RoboDK station: 6640_station_curve1.rdk

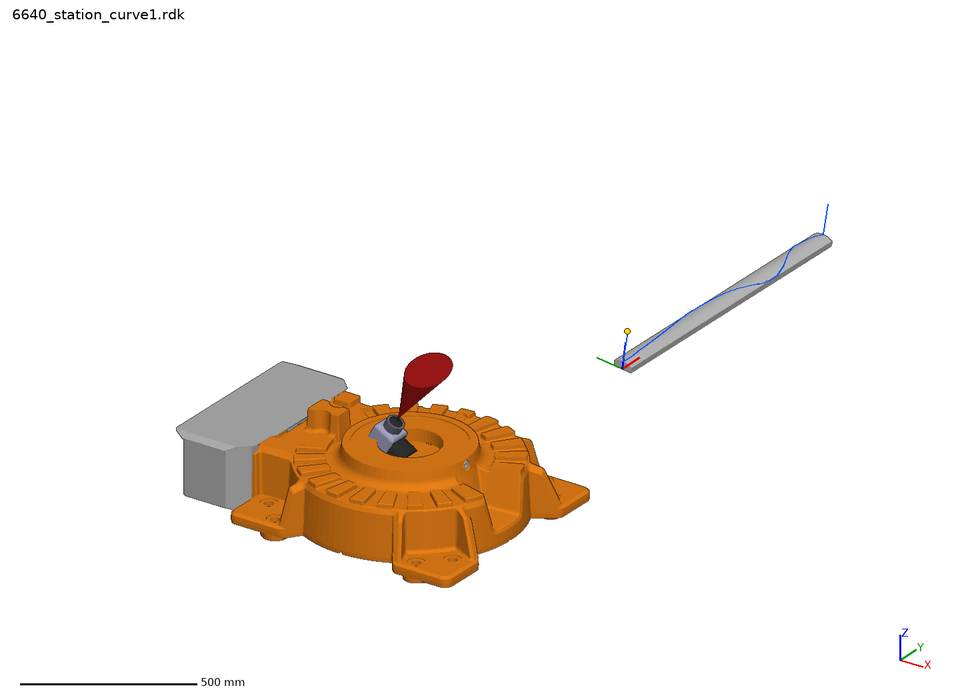
[picture v0: the station drawn from its stored meshes, robots at their saved joint values, targets as dots, program paths as lines]
Station 6640_station_curve1 (saved by RoboDK 5.3.2). Poses are relative to the parent item; angles as X-Y-Z fixed-axis rotations.
  - frame Frame 3 at (1086.51, -506.82, 968.91) mm, rotated rx 8.27 ry 0.16 rz 90.47 deg
    - object Curve_sparse at (0, 0, 0) mm
    - object wood at (0, 0, 0) mm, size 1000 x 60 x 25.4 mm, geometry from wood.stl
  - machining project Path1 settings: rotZ(0) | rotX(0)*rotY(0) | rotz(0)
  - program Path1 (113 instructions, listed below)
  - robot ABB IRB 6640-180/2.55: 6 axes, payload 180 kg, reach 2550 mm, repeatability 0.07 mm, weight 1310 kg
      joint limits [-170, -65, -180, -300, -120, -360] to [170, 85, 70, 300, 120, 360]; home [0, 0, 0, 0, 0, 0]; saved at [28.636, -24.413, 34.192, -11.874, 61.538, 32.546]
    - tool Paint gun, TCP at (75, 0, 493.3) mm, rotated rx 0 ry 30 rz 0 deg, size 203.2 x 279.7 x 471.5 mm
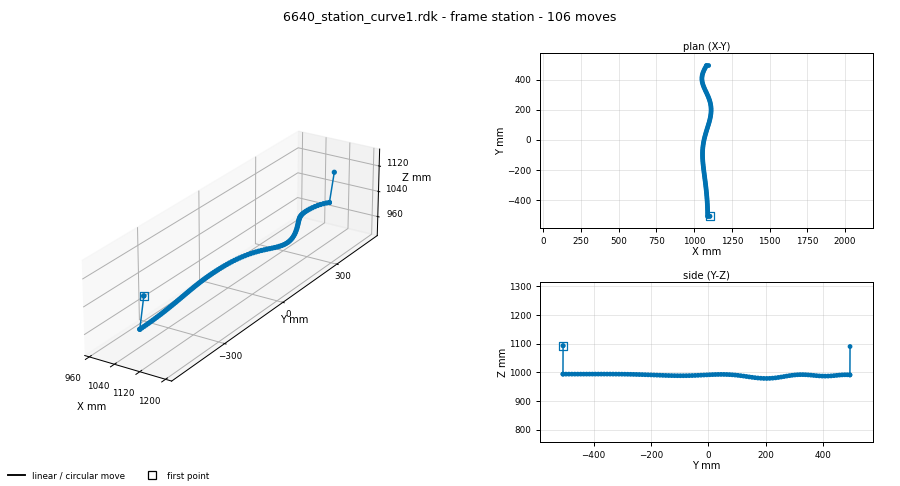
[picture p0: tool path of 6640_station_curve1.rdk in frame station, 106 of 106 moves have a stored position in this frame; points joined in program order, loops and branches not executed]

--- program Path1 (robot ABB IRB 6640-180/2.55) ---
  Smooth(1)
  Set speed (500.0 mm/s)
  Set Ref.: Frame 3
  Set Tool: Paint gun
  Show Paint gun
  MoveJ 1 to (0, 0, 125.4) mm, rotated rx 180 ry 0 rz 89.52 deg; joints [-28.763, -23.766, 33.648, 11.507, 61.252, -32.677]
  MoveL 2 to (0, 0, 125.4) mm, rotated rx 180 ry 0 rz 89.52 deg; joints [-28.763, -23.766, 33.648, 11.507, 61.252, -32.677]
  MoveL 3 to (0, 0, 25.4) mm, rotated rx 180 ry 0 rz 89.52 deg; joints [-29.166, -24.266, 38.853, 12.236, 56.729, -34.255]
  MoveL 4 to (0, 0, 25.4) mm, rotated rx 180 ry 0 rz 89.52 deg; joints [-29.166, -24.266, 38.853, 12.236, 56.729, -34.255]
  Set speed (50.0 mm/s)
  MoveL 5 to (10.27, 0.03, 25.4) mm, rotated rx 180 ry 0.03 rz 89.52 deg; joints [-28.68, -24.594, 39.061, 12.062, 56.719, -33.688]
  MoveL 6 to (20.55, 0.12, 25.4) mm, rotated rx 180 ry 0.13 rz 89.52 deg; joints [-28.212, -24.963, 39.304, 11.937, 56.664, -33.163]
  MoveL 7 to (30.82, 0.27, 25.4) mm, rotated rx 180 ry 0.3 rz 89.52 deg; joints [-27.761, -25.373, 39.58, 11.859, 56.565, -32.678]
  MoveL 8 to (41.1, 0.48, 25.4) mm, rotated rx 180 ry 0.54 rz 89.52 deg; joints [-27.327, -25.825, 39.89, 11.827, 56.42, -32.233]
  MoveL 9 to (51.37, 0.75, 25.39) mm, rotated rx 179.99 ry 0.84 rz 89.52 deg; joints [-26.908, -26.32, 40.233, 11.838, 56.23, -31.825]
  MoveL 10 to (61.65, 1.07, 25.39) mm, rotated rx 179.99 ry 1.21 rz 89.52 deg; joints [-26.505, -26.859, 40.611, 11.891, 55.993, -31.454]
  MoveL 11 to (71.92, 1.46, 25.38) mm, rotated rx 179.99 ry 1.65 rz 89.52 deg; joints [-26.116, -27.442, 41.023, 11.986, 55.711, -31.119]
  MoveL 12 to (82.18, 1.91, 25.36) mm, rotated rx 179.98 ry 2.15 rz 89.52 deg; joints [-25.741, -28.07, 41.469, 12.121, 55.383, -30.819]
  MoveL 13 to (92.45, 2.41, 25.34) mm, rotated rx 179.98 ry 2.72 rz 89.52 deg; joints [-25.379, -28.743, 41.949, 12.295, 55.009, -30.552]
  MoveL 14 to (102.71, 2.98, 25.31) mm, rotated rx 179.97 ry 3.35 rz 89.52 deg; joints [-25.03, -29.461, 42.464, 12.507, 54.591, -30.32]
  MoveL 15 to (112.97, 3.6, 25.27) mm, rotated rx 179.97 ry 4.05 rz 89.52 deg; joints [-24.692, -30.224, 43.013, 12.756, 54.127, -30.119]
  MoveL 16 to (123.22, 4.28, 25.22) mm, rotated rx 179.96 ry 4.81 rz 89.52 deg; joints [-24.365, -31.033, 43.595, 13.042, 53.621, -29.95]
  MoveL 17 to (133.47, 5.01, 25.15) mm, rotated rx 179.95 ry 5.64 rz 89.52 deg; joints [-24.047, -31.886, 44.21, 13.362, 53.072, -29.811]
  MoveL 18 to (143.72, 5.8, 25.07) mm, rotated rx 179.95 ry 6.52 rz 89.52 deg; joints [-23.737, -32.783, 44.857, 13.716, 52.483, -29.701]
  MoveL 19 to (153.96, 6.65, 24.97) mm, rotated rx 179.94 ry 7.45 rz 89.52 deg; joints [-23.435, -33.723, 45.536, 14.101, 51.854, -29.619]
  MoveL 20 to (164.2, 7.54, 24.84) mm, rotated rx 179.93 ry 8.44 rz 89.52 deg; joints [-23.137, -34.705, 46.244, 14.515, 51.19, -29.561]
  MoveL 21 to (174.44, 8.49, 24.69) mm, rotated rx 179.92 ry 9.48 rz 89.52 deg; joints [-22.843, -35.726, 46.981, 14.956, 50.491, -29.527]
  MoveL 22 to (184.66, 9.48, 24.52) mm, rotated rx 179.91 ry 10.57 rz 89.52 deg; joints [-22.55, -36.783, 47.743, 15.421, 49.762, -29.511]
  MoveL 23 to (194.89, 10.51, 24.31) mm, rotated rx 179.9 ry 11.69 rz 89.51 deg; joints [-22.256, -37.875, 48.528, 15.904, 49.006, -29.511]
  MoveL 24 to (205.11, 11.59, 24.08) mm, rotated rx 179.89 ry 12.85 rz 89.51 deg; joints [-21.959, -38.997, 49.334, 16.402, 48.225, -29.522]
  MoveL 25 to (215.32, 12.7, 23.81) mm, rotated rx 179.88 ry 14.03 rz 89.51 deg; joints [-21.654, -40.146, 50.156, 16.908, 47.426, -29.538]
  MoveL 26 to (225.53, 13.84, 23.52) mm, rotated rx 179.87 ry 15.24 rz 89.5 deg; joints [-21.34, -41.317, 50.991, 17.415, 46.611, -29.552]
  MoveL 27 to (235.73, 15, 23.18) mm, rotated rx 179.86 ry 16.45 rz 89.5 deg; joints [-21.012, -42.505, 51.834, 17.916, 45.786, -29.557]
  MoveL 28 to (245.94, 16.19, 22.82) mm, rotated rx 179.85 ry 17.68 rz 89.5 deg; joints [-20.667, -43.704, 52.681, 18.4, 44.955, -29.543]
  MoveL 29 to (256.14, 17.39, 22.42) mm, rotated rx 179.83 ry 18.9 rz 89.49 deg; joints [-20.301, -44.909, 53.526, 18.858, 44.122, -29.502]
  MoveL 30 to (266.33, 18.6, 22) mm, rotated rx 179.82 ry 20.1 rz 89.48 deg; joints [-19.91, -46.112, 54.365, 19.278, 43.293, -29.422]
  MoveL 31 to (276.53, 19.8, 21.54) mm, rotated rx 179.81 ry 21.29 rz 89.48 deg; joints [-19.49, -47.308, 55.191, 19.646, 42.473, -29.291]
  MoveL 32 to (286.73, 20.99, 21.06) mm, rotated rx 179.8 ry 22.45 rz 89.47 deg; joints [-19.036, -48.488, 55.998, 19.951, 41.665, -29.097]
  MoveL 33 to (296.93, 22.16, 20.57) mm, rotated rx 179.79 ry 23.56 rz 89.46 deg; joints [-18.546, -49.644, 56.78, 20.176, 40.876, -28.827]
  MoveL 34 to (307.13, 23.29, 20.06) mm, rotated rx 179.77 ry 24.63 rz 89.46 deg; joints [-18.015, -50.768, 57.531, 20.307, 40.109, -28.466]
  MoveL 35 to (317.34, 24.39, 19.55) mm, rotated rx 179.76 ry 25.64 rz 89.45 deg; joints [-17.44, -51.851, 58.245, 20.331, 39.37, -28.002]
  MoveL 36 to (327.55, 25.42, 19.04) mm, rotated rx 179.75 ry 26.59 rz 89.44 deg; joints [-16.818, -52.883, 58.914, 20.231, 38.664, -27.422]
  MoveL 37 to (337.77, 26.39, 18.54) mm, rotated rx 179.74 ry 27.45 rz 89.43 deg; joints [-16.146, -53.855, 59.534, 19.995, 37.996, -26.713]
  MoveL 38 to (348, 27.28, 18.08) mm, rotated rx 179.73 ry 28.23 rz 89.43 deg; joints [-15.422, -54.756, 60.096, 19.611, 37.374, -25.864]
  MoveL 39 to (358.24, 28.06, 17.65) mm, rotated rx 179.72 ry 28.92 rz 89.42 deg; joints [-14.647, -55.574, 60.594, 19.07, 36.803, -24.867]
  MoveL 40 to (368.48, 28.74, 17.27) mm, rotated rx 179.71 ry 29.5 rz 89.41 deg; joints [-13.819, -56.299, 61.021, 18.363, 36.293, -23.717]
  MoveL 41 to (378.74, 29.28, 16.96) mm, rotated rx 179.71 ry 29.96 rz 89.41 deg; joints [-12.939, -56.917, 61.371, 17.488, 35.851, -22.41]
  MoveL 42 to (389.01, 29.69, 16.73) mm, rotated rx 179.7 ry 30.3 rz 89.41 deg; joints [-12.01, -57.416, 61.637, 16.448, 35.489, -20.948]
  MoveL 43 to (399.28, 29.93, 16.58) mm, rotated rx 179.7 ry 30.5 rz 89.4 deg; joints [-11.036, -57.782, 61.81, 15.249, 35.219, -19.34]
  MoveL 44 to (409.55, 30, 16.54) mm, rotated rx 179.7 ry 30.56 rz 89.4 deg; joints [-10.021, -58.003, 61.885, 13.906, 35.051, -17.599]
  MoveL 45 to (419.82, 29.88, 16.61) mm, rotated rx 179.7 ry 30.46 rz 89.41 deg; joints [-8.971, -58.064, 61.852, 12.439, 35, -15.743]
  MoveL 46 to (430.09, 29.55, 16.8) mm, rotated rx 179.7 ry 30.19 rz 89.41 deg; joints [-7.893, -57.953, 61.705, 10.874, 35.08, -13.798]
  MoveL 47 to (440.35, 29.02, 17.11) mm, rotated rx 179.71 ry 29.73 rz 89.41 deg; joints [-6.798, -57.657, 61.436, 9.247, 35.305, -11.795]
  MoveL 48 to (450.59, 28.26, 17.54) mm, rotated rx 179.72 ry 29.08 rz 89.42 deg; joints [-5.695, -57.164, 61.038, 7.597, 35.69, -9.772]
  MoveL 49 to (460.8, 27.26, 18.08) mm, rotated rx 179.73 ry 28.22 rz 89.43 deg; joints [-4.595, -56.464, 60.503, 5.966, 36.248, -7.769]
  MoveL 50 to (470.99, 26.04, 18.73) mm, rotated rx 179.74 ry 27.14 rz 89.44 deg; joints [-3.511, -55.548, 59.823, 4.398, 36.992, -5.826]
  MoveL 51 to (481.13, 24.57, 19.46) mm, rotated rx 179.76 ry 25.81 rz 89.45 deg; joints [-2.455, -54.409, 58.994, 2.935, 37.931, -3.981]
  MoveL 52 to (491.24, 22.88, 20.25) mm, rotated rx 179.78 ry 24.24 rz 89.46 deg; joints [-1.438, -53.042, 58.011, 1.613, 39.076, -2.269]
  MoveL 53 to (501.3, 20.95, 21.08) mm, rotated rx 179.8 ry 22.41 rz 89.47 deg; joints [-0.471, -51.445, 56.869, 0.461, 40.433, -0.718]
  MoveL 54 to (511.32, 18.81, 21.92) mm, rotated rx 179.82 ry 20.31 rz 89.48 deg; joints [0.435, -49.618, 55.569, -0.501, 42.005, 0.656]
  MoveL 55 to (521.29, 16.45, 22.74) mm, rotated rx 179.84 ry 17.95 rz 89.49 deg; joints [1.274, -47.568, 54.113, -1.264, 43.792, 1.842]
  MoveL 56 to (531.21, 13.91, 23.5) mm, rotated rx 179.87 ry 15.31 rz 89.5 deg; joints [2.039, -45.304, 52.508, -1.827, 45.788, 2.841]
  MoveL 57 to (541.1, 11.19, 24.17) mm, rotated rx 179.9 ry 12.42 rz 89.51 deg; joints [2.729, -42.844, 50.769, -2.202, 47.981, 3.663]
  MoveL 58 to (550.95, 8.31, 24.72) mm, rotated rx 179.92 ry 9.29 rz 89.52 deg; joints [3.344, -40.212, 48.912, -2.407, 50.351, 4.325]
  MoveL 59 to (560.77, 5.31, 25.12) mm, rotated rx 179.95 ry 5.96 rz 89.52 deg; joints [3.888, -37.44, 46.967, -2.465, 52.868, 4.848]
  MoveL 60 to (570.57, 2.2, 25.35) mm, rotated rx 179.98 ry 2.48 rz 89.52 deg; joints [4.366, -34.57, 44.964, -2.402, 55.495, 5.259]
  MoveL 61 to (580.34, -0.98, 25.39) mm, rotated rx -179.99 ry -1.1 rz 89.52 deg; joints [4.789, -31.65, 42.942, -2.246, 58.183, 5.584]
  MoveL 62 to (590.1, -4.2, 25.23) mm, rotated rx -179.96 ry -4.72 rz 89.51 deg; joints [5.165, -28.732, 40.94, -2.022, 60.883, 5.846]
  MoveL 63 to (599.85, -7.41, 24.86) mm, rotated rx -179.93 ry -8.3 rz 89.5 deg; joints [5.506, -25.87, 39, -1.753, 63.536, 6.068]
  MoveL 64 to (609.6, -10.59, 24.3) mm, rotated rx -179.89 ry -11.78 rz 89.48 deg; joints [5.821, -23.114, 37.155, -1.457, 66.093, 6.268]
  MoveL 65 to (619.37, -13.69, 23.55) mm, rotated rx -179.86 ry -15.08 rz 89.46 deg; joints [6.122, -20.509, 35.436, -1.148, 68.506, 6.46]
  MoveL 66 to (629.17, -16.67, 22.66) mm, rotated rx -179.83 ry -18.17 rz 89.44 deg; joints [6.415, -18.095, 33.866, -0.838, 70.734, 6.655]
  MoveL 67 to (639.01, -19.48, 21.66) mm, rotated rx -179.79 ry -20.98 rz 89.42 deg; joints [6.709, -15.901, 32.46, -0.535, 72.747, 6.861]
  MoveL 68 to (648.9, -22.07, 20.6) mm, rotated rx -179.76 ry -23.49 rz 89.39 deg; joints [7.008, -13.952, 31.228, -0.246, 74.52, 7.085]
  MoveL 69 to (658.85, -24.39, 19.54) mm, rotated rx -179.73 ry -25.65 rz 89.37 deg; joints [7.32, -12.263, 30.174, 0.025, 76.036, 7.329]
  MoveL 70 to (668.88, -26.39, 18.55) mm, rotated rx -179.7 ry -27.45 rz 89.34 deg; joints [7.647, -10.852, 29.3, 0.271, 77.285, 7.599]
  MoveL 71 to (679, -28, 17.68) mm, rotated rx -179.67 ry -28.86 rz 89.32 deg; joints [7.995, -9.73, 28.609, 0.488, 78.253, 7.898]
  MoveL 72 to (689.18, -29.17, 17.03) mm, rotated rx -179.65 ry -29.86 rz 89.3 deg; joints [8.367, -8.911, 28.103, 0.669, 78.931, 8.23]
  MoveL 73 to (699.43, -29.84, 16.63) mm, rotated rx -179.64 ry -30.43 rz 89.29 deg; joints [8.769, -8.409, 27.786, 0.807, 79.306, 8.6]
  MoveL 74 to (709.7, -29.98, 16.55) mm, rotated rx -179.64 ry -30.55 rz 89.29 deg; joints [9.204, -8.24, 27.664, 0.891, 79.366, 9.014]
  MoveL 75 to (719.96, -29.55, 16.8) mm, rotated rx -179.65 ry -30.19 rz 89.3 deg; joints [9.679, -8.417, 27.747, 0.909, 79.097, 9.481]
  MoveL 76 to (730.17, -28.55, 17.38) mm, rotated rx -179.66 ry -29.33 rz 89.31 deg; joints [10.201, -8.953, 28.045, 0.846, 78.484, 10.012]
  MoveL 77 to (740.29, -26.98, 18.24) mm, rotated rx -179.69 ry -27.97 rz 89.33 deg; joints [10.777, -9.859, 28.571, 0.684, 77.512, 10.621]
  MoveL 78 to (750.29, -24.88, 19.31) mm, rotated rx -179.72 ry -26.09 rz 89.36 deg; joints [11.421, -11.141, 29.34, 0.399, 76.168, 11.329]
  MoveL 79 to (760.16, -22.28, 20.51) mm, rotated rx -179.75 ry -23.68 rz 89.39 deg; joints [12.145, -12.806, 30.368, -0.037, 74.441, 12.164]
  MoveL 80 to (769.9, -19.25, 21.75) mm, rotated rx -179.79 ry -20.75 rz 89.42 deg; joints [12.97, -14.851, 31.669, -0.664, 72.325, 13.163]
  MoveL 81 to (779.52, -15.84, 22.93) mm, rotated rx -179.84 ry -17.32 rz 89.45 deg; joints [13.916, -17.268, 33.255, -1.53, 69.825, 14.376]
  MoveL 82 to (789.04, -12.11, 23.96) mm, rotated rx -179.88 ry -13.41 rz 89.47 deg; joints [15.007, -20.03, 35.127, -2.698, 66.968, 15.865]
  MoveL 83 to (798.48, -8.12, 24.75) mm, rotated rx -179.92 ry -9.08 rz 89.5 deg; joints [16.266, -23.089, 37.271, -4.242, 63.807, 17.704]
  MoveL 84 to (807.86, -3.95, 25.25) mm, rotated rx -179.96 ry -4.45 rz 89.51 deg; joints [17.711, -26.369, 39.65, -6.246, 60.432, 19.977]
  MoveL 85 to (817.21, 0.33, 25.4) mm, rotated rx 180 ry 0.37 rz 89.52 deg; joints [19.348, -29.766, 42.205, -8.789, 56.971, 22.761]
  MoveL 86 to (826.53, 4.64, 25.19) mm, rotated rx 179.96 ry 5.22 rz 89.52 deg; joints [21.165, -33.153, 44.853, -11.93, 53.584, 26.114]
  MoveL 87 to (835.86, 8.91, 24.62) mm, rotated rx 179.92 ry 9.95 rz 89.52 deg; joints [23.131, -36.401, 47.499, -15.677, 50.439, 30.044]
  MoveL 88 to (845.23, 13.05, 23.72) mm, rotated rx 179.88 ry 14.4 rz 89.51 deg; joints [25.194, -39.389, 50.048, -19.958, 47.69, 34.483]
  MoveL 89 to (854.66, 16.97, 22.57) mm, rotated rx 179.84 ry 18.47 rz 89.49 deg; joints [27.285, -42.018, 52.412, -24.611, 45.447, 39.277]
  MoveL 90 to (864.19, 20.57, 21.24) mm, rotated rx 179.8 ry 22.04 rz 89.47 deg; joints [29.332, -44.217, 54.517, -29.387, 43.76, 44.191]
  MoveL 91 to (873.86, 23.76, 19.85) mm, rotated rx 179.77 ry 25.06 rz 89.45 deg; joints [31.262, -45.942, 56.301, -33.982, 42.615, 48.942]
  MoveL 92 to (883.7, 26.41, 18.53) mm, rotated rx 179.74 ry 27.47 rz 89.43 deg; joints [33.007, -47.168, 57.715, -38.088, 41.948, 53.24]
  MoveL 93 to (893.72, 28.42, 17.45) mm, rotated rx 179.72 ry 29.22 rz 89.42 deg; joints [34.506, -47.883, 58.712, -41.421, 41.661, 56.819]
  MoveL 94 to (903.9, 29.65, 16.75) mm, rotated rx 179.7 ry 30.27 rz 89.41 deg; joints [35.7, -48.084, 59.247, -43.747, 41.651, 59.458]
  MoveL 95 to (914.16, 29.99, 16.55) mm, rotated rx 179.7 ry 30.56 rz 89.4 deg; joints [36.539, -47.778, 59.286, -44.889, 41.834, 60.989]
  MoveL 96 to (924.4, 29.4, 16.89) mm, rotated rx 179.7 ry 30.06 rz 89.41 deg; joints [36.989, -46.979, 58.807, -44.751, 42.158, 61.31]
  MoveL 97 to (934.53, 27.89, 17.74) mm, rotated rx 179.72 ry 28.77 rz 89.42 deg; joints [37.034, -45.706, 57.809, -43.315, 42.629, 60.396]
  MoveL 98 to (944.45, 25.53, 18.98) mm, rotated rx 179.75 ry 26.68 rz 89.44 deg; joints [36.68, -43.978, 56.308, -40.653, 43.303, 58.307]
  MoveL 99 to (954.14, 22.43, 20.45) mm, rotated rx 179.78 ry 23.82 rz 89.46 deg; joints [35.955, -41.805, 54.335, -36.924, 44.286, 55.187]
  MoveL 100 to (963.6, 18.71, 21.95) mm, rotated rx 179.82 ry 20.22 rz 89.48 deg; joints [34.902, -39.191, 51.928, -32.366, 45.707, 51.264]
  MoveL 101 to (972.87, 14.5, 23.33) mm, rotated rx 179.86 ry 15.93 rz 89.5 deg; joints [33.587, -36.144, 49.141, -27.3, 47.68, 46.847]
  MoveL 102 to (982, 9.9, 24.44) mm, rotated rx 179.91 ry 11.03 rz 89.52 deg; joints [32.095, -32.696, 46.05, -22.092, 50.267, 42.294]
  MoveL 103 to (991.02, 5.03, 25.15) mm, rotated rx 179.95 ry 5.66 rz 89.52 deg; joints [30.529, -28.921, 42.761, -17.097, 53.433, 37.956]
  MoveL 104 to (999.96, 0.02, 25.4) mm, rotated rx 180 ry 0.02 rz 89.52 deg; joints [29.002, -24.948, 39.414, -12.595, 57.034, 34.108]
  Set speed (500.0 mm/s)
  MoveL 105 to (999.96, 0.02, 25.4) mm, rotated rx 180 ry 0.02 rz 89.52 deg; joints [29.002, -24.948, 39.414, -12.595, 57.034, 34.108]
  MoveL 106 to (999.96, 0.06, 125.4) mm, rotated rx 180 ry 0.02 rz 89.52 deg; joints [28.636, -24.413, 34.192, -11.874, 61.538, 32.546]
